// TIA Portal project "Elevator Emergency Stop" (V17)
// Elevator Emergency Stop
// When the Emergency button is pressed, stop the elevator immediately. Open the doors once stopped.
// When Reset button is pressed, it clears the faults, i.e., the doors will close and the elevator will start again

(* hardware
DEVICE "S7-1200 station_1"  S7-1200 Station
   slot 0: "Rack_0"  S7-1200 Rack  Rack  V1.0
   slot 1: "PLC_1"  CPU 1215C AC/DC/Rly  6ES7 215-1BG40-0XB0  V4.5
*)

// ===== PLC "PLC_1"  CPU 1215C AC/DC/Rly =====

VAR_GLOBAL   // PLC tag table "Default tag table"
   "Emergency" AT %I0.0 : Bool;
   "Switch ON" AT %I0.1 : Bool;
   "Reset" AT %I0.2 : Bool;
   "Elevator" AT %Q0.0 : Bool;
   "Door" AT %Q0.1 : Bool;
   "Tag_1" AT %M0.0 : Bool;
   "Tag_2" AT %M0.1 : Bool;
END_VAR

ORGANIZATION_BLOCK "Main"   // OB1, LAD, ProgramCycle
TITLE = "Main Program Sweep (Cycle)"
{ S7_Optimized_Access := 'TRUE' }
VERSION : 0.1
   VAR_INPUT
      Initial_Call : Bool;   // Initial call of this OB
      Remanence : Bool;   // =True, if remanent data are available
   END_VAR
BEGIN

REGION Network 1
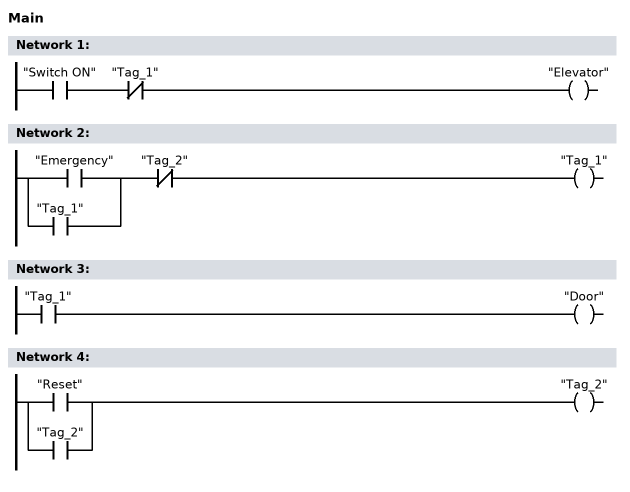
   RUNG wire#powerrail
      Contact( "Switch ON" )
      I_Contact( "Tag_1" )
      Coil( "Elevator" )
   END_RUNG
   // the same network as SCL:
   "Elevator" := "Switch ON" AND NOT "Tag_1";
END_REGION

REGION Network 2
   RUNG wire#powerrail
      Contact( "Emergency" )
      wire#w1
      I_Contact( "Tag_2" )
      Coil( "Tag_1" )
   END_RUNG
   RUNG wire#powerrail
      Contact( "Tag_1" )
   END_RUNG wire#w1
   // the same network as SCL:
   "Tag_1" := ("Emergency" OR "Tag_1") AND NOT "Tag_2";
END_REGION

REGION Network 3
   RUNG wire#powerrail
      Contact( "Tag_1" )
      Coil( "Door" )
   END_RUNG
   // the same network as SCL:
   "Door" := "Tag_1";
END_REGION

REGION Network 4
   RUNG wire#powerrail
      Contact( "Reset" )
      wire#w1
      Coil( "Tag_2" )
   END_RUNG
   RUNG wire#powerrail
      Contact( "Tag_2" )
   END_RUNG wire#w1
   // the same network as SCL:
   "Tag_2" := "Reset" OR "Tag_2";
END_REGION
END_ORGANIZATION_BLOCK